FUNCTION F_GetCheckSumByte : BYTE
VAR_INPUT
	aData: ARRAY[0..30] OF BYTE;
	nLength: USINT;
END_VAR
VAR
	i: USINT;
	nTemp: BYTE;
END_VAR

FOR i:= 0 TO nLength-1 BY 1 DO
	nTemp := aData[i] XOR nTemp;
END_FOR

F_GetCheckSumByte := nTemp;

END_FUNCTION

(* stored: Version 1.1.0.1, ProductVersion 3.1.0.25
   POU F_GetCheckSumByte: Id {424547fe-e718-4843-ab5d-f44b15df7b19} *)
